# EPICS autosave request: iocBoot/commonSettings.req
$(P):CAL:CH1
$(P):CAL:CH4
$(P):UNITS:P:CH1
$(P):UNITS:P:CH4
$(P):UNITS:T:CH1
$(P):UNITS:T:CH4
$(P):DIS:CH4
$(P):SEQ:CH1:1.SCAN
